PROGRAM MAIN
VAR
	
	queue : Queue;
	size : UINT;
	
	// showing the use of the queue for the same datatype
	trigger : BOOL;
	position1 : Coordinate3D :=  (x:=3, y:=8, z:=-1);
	position2 : Coordinate3D :=  (x:=9, y:=1, z:=0);
	currentPosition : Coordinate3D;
	
	// showing the same queue can be used for anything at any time!
	trigger2 : BOOL;	
	myInt : INT := 123;
	myBool : BOOL := TRUE;
	myPosition : Coordinate3D :=  (x:=3, y:=8, z:=-1);
	poppedInt : INT;
	poppedBool : BOOL;
	poppedPosition : Coordinate3D;	
	
END_VAR

// example showing the queue can hold any number of the same type. 
IF trigger THEN
	
	trigger := FALSE;
	
	queue.Push(position1);
	queue.Push(position2);
	
	size := queue.Size(); // size 2
	queue.Pop(currentPosition); // (x:=3, y:=8, z:=-1)
	size := queue.Size(); // size 1
	queue.Pop(currentPosition); // (x:=9, y:=1, z:=0)
	size := queue.Size(); // size 0

END_IF

// example showing the queue can hold any number of any type all at the same time. 
IF trigger2 THEN
	
	trigger2 := FALSE;
	
	queue.Push(myInt);
	queue.Push(myBool);
	queue.Push(myPosition);
	
	size := queue.Size(); // size 3
	queue.Pop(poppedBool); // The datatype is wrong as the first push was an INT so nothing is popped.
	
	size := queue.Size(); // size 3
	queue.Pop(poppedInt); // 123
	size := queue.Size(); // size 2
	queue.Pop(poppedBool); // true
	size := queue.Size(); // size 1
	queue.Pop(poppedPosition); // (x:=3, y:=8, z:=-1)
	size := queue.Size(); // size 0
	
END_IF

END_PROGRAM

(* stored: Version 1.1.0.1, ProductVersion 3.1.4024.11
   POU MAIN: Id {d764e607-8c77-441b-9951-16fc2e18c7ff}, SpecialFunc None *)
